(*
  This StartPosDetect supports different modes:
  - Triangle Markus
  - Internal StartPos generation (simulation based on substrate length and gap)
*)
FUNCTION_BLOCK FB_StartPositionWeu EXTENDS T_NamedBase IMPLEMENTS I_StartPosDetect
VAR_INPUT
  bEnable                         : BOOL;            // enable start position detection
  nCurrentPos                     : DINT;            // current position in Pulses/Subpixels
  fCurrentSpeed                   : LREAL;           // actual speed of conveyor in [m/s]
  fSubstrateLength                : LREAL;           // substrate length in [m]
  bUseExternalStartPos            : BOOL;            // Use external start position source
END_VAR
VAR_OUTPUT
  fLateralOffset                  : LREAL;           // Lateral +/- shift in Y [m]
  fSubstrateLengthDetected        : LREAL;           // Detected substrate length
  nPrintMarkPosBits               : WORD;            // Print mark position (bit coded),  TODO: avoid this specific code
END_VAR
VAR
  bInit : BOOL;   // fb initialized
  nMode : (MARK, SIMULATE_INTERN, SIMULATE_EXTERN) := MARK;   // StartTrigger mode
  
  // config
  _fResolutionPrint : LREAL;
  _fResolutionSubPx : LREAL;
  _pMarkDefinition : POINTER TO ST_MarkDefinition_Triangle;
  _iStartPosDetectExt : I_StartPosDetect;   // external start position source
   
  // instances
  fbMarkDetection : FB_MarkDetection_Triangle;    // StartPosition detection by marks
  fbStartPosSim   : FB_StartPositionDummy;        // StartPosition simulation

  // helper
  _bStart : BOOL;
  _nX0 : DINT;
  _bValid : BOOL;
  tOn_MissingMarksCheck : TON;   // trigger check (triggers within given time)
END_VAR

// TODO: >>>>>>>>>>>>>>>>>>>>>>>>>>>>>>>>>>>
// (optional) Mode: Encoder C HW_LATCH instead of marks
// <<<<<<<<<<<<<<<<<<<<<<<<<<<<<<<<<<<<<<<<<

// check parameter
IF NOT bInit THEN RETURN; END_IF
IF fCurrentSpeed = 0 THEN RETURN ; END_IF   // avoid 0 division

// default values (outputs and properties)
_bStart := FALSE;
_bValid := TRUE;
nPrintMarkPosBits := 0;  // no marks used
fLateralOFfset := 0;
fSubstrateLengthDetected := fSubstrateLength;

// mode selection
IF _pMarkDefinition = 0 OR_ELSE NOT _pMarkDefinition^.bEnabled THEN
  nMode :=  SEL(bUseExternalStartPos AND _iStartPosDetectExt <> 0, 
                  SIMULATE_INTERN, 
                  SIMULATE_EXTERN
                );
ELSIF NOT _pMarkDefinition^.bEnabled THEN   // if mark config is given and enabled
  nMode := MARK; 
END_IF

// run mode
IF nMode = MARK  THEN 
  // - with mark (forward / backward / other mark orientation)
  fbMarkDetection(
    bEnable:=bEnable,
    fResolution:=_fResolutionPrint*_fResolutionSubPx,
    fSubstrateLength:=fSubstrateLength,
    pMarkDefinition:=_pMarkDefinition,
    nCurrentPos:=nCurrentPos,
    fCurrentSpeed:=fCurrentSpeed,
    //bStartTrig=>_bStart,
    //nOffset_X0=>_nX0,
    fLateralOffset=>fLateralOffset,
    fSubstrateLengthDetected=>fSubstrateLengthDetected
  );
  // set I_StartPosDetect properties
  _bStart := fbMarkDetection.bStartTrig;
  _bValid := TRUE;
  _nX0    := fbMarkDetection.nOffset_X0;
  
 (*Check area with the correct arrangement of the mark sensor*)
 IF fbMarkDetection.bAreaOk THEN nPrintMarkPosBits.2 := TRUE; (*mark position in center*) 
  ELSIF fbMarkDetection.fLateralOffset > 0  THEN nPrintMarkPosBits.1 := TRUE; (*mark position on side I*) 
  ELSIF fbMarkDetection.fLateralOffset < 0  THEN nPrintMarkPosBits.3 := TRUE; (*mark position on side II*) 
  END_IF
  
  
ELSIF nMode = SIMULATE_INTERN THEN
  // without mark, simulate internally, started by external trigger and re-occur after every image/sheet length
  fbStartPosSim.bEnable := bEnable;                     // start simulatin with enable
  fbStartPosSim.bAutoTrigger := TRUE;
  fbStartPosSim.fSheetGap := 0;
  fbStartPosSim.fSubstrateLength := fSubstrateLength;   // same as given
  fbStartPosSim(
    //bTrigger:=,
    lPosition:=nCurrentPos,
    fSpeed:=fCurrentSpeed,
    fResolution:=_fResolutionPrint*_fResolutionSubPx
  );
  // set I_StartPosDetect properties
  _bStart := fbStartPosSim.bStartTrig;
  _bValid := fbStartPosSim.bValid;
  _nX0    := fbStartPosSim.nStartPositionX0;
  
  
ELSIF nMode = SIMULATE_EXTERN THEN
  // without mark, based on external reference
  
  // set I_StartPosDetect properties
  _bStart := ;
  _bValid := TRUE;
  _nX0    := ;
ELSE
  ;
END_IF


// supervision of mark missing (at least one trigger within 2 image lengths
//     nPrintMarkPosBits.0 := TRUE; (*=1 mark missing*) 
tOn_MissingMarksCheck(IN := bEnable AND NOT _bStart, PT := REAL_TO_TIME((2 * fSubstrateLength) / fCurrentSpeed * 1000), 
                      Q=>nPrintMarkPosBits.0
);

{warning 'add property implementation'}
(*
  A new container detected.
  NOTE: a pulse only
*)
PROPERTY bStartTrig : BOOL
GET
bStartTrig := _bStart;
END_GET
END_PROPERTY

{warning 'add property implementation'}
(*
  A valid container detected.
*)
PROPERTY bValid : BOOL
GET
bValid := _bValid;
END_GET
END_PROPERTY

METHOD Init
VAR_INPUT
  fPrintResolution      : LREAL := 600;         // print(head) resolution in [dpi]
  fSubPxResolution      : LREAL := 32;          // SubPixel resolution [SubPx], resolution factor (fI_PrintResolution*fI_SubPxResolution=>Output resolution)
  pMarkDefinition       : POINTER TO ST_MarkDefinition_Triangle;
  iStartPosDetectExt     : I_StartPosDetect;   // external start position source
END_VAR
IF _pMarkDefinition = 0 THEN LogError('Invalid parameter'); END_IF

_fResolutionPrint := fPrintResolution;
_fResolutionSubPx := fSubPxResolution;
_pMarkDefinition := pMarkDefinition;
_iStartPosDetectExt := iStartPosDetectExt;

// (optional) we use pointerTo_PU.registerStatusClient(sClient := fbStartPosSim);

bInit := TRUE;
END_METHOD

{warning 'add property implementation'}
(*
  Detected start position X0 (absolute) in [SubPx].
*)
PROPERTY nStartPositionX0 : DINT
GET
nStartPositionX0 := _nX0;
END_GET
END_PROPERTY

METHOD reset
fbMarkDetection.reset();
END_METHOD

END_FUNCTION_BLOCK

(* stored: Version 1.1.0.1, ProductVersion 3.1.4024.11
   POU FB_StartPositionWeu: Id {57e46adf-0651-4188-b0a4-ce8ff8a13827}, SpecialFunc None
   Folder I_StartPosDetect: Id {3bb3d753-1c9e-472a-8c3f-aec14f002339}
   Property bStartTrig: Id {e283e51a-7bd3-43b7-929a-8344709bc1e4}
   Get Get: Id {d88d396b-d2d9-47aa-81b3-e6702f1b2da2}
   Property bValid: Id {41d06b7b-92f2-4bfb-b40f-9ec4299b6723}
   Get Get: Id {b92c99f7-0a7d-43bc-bf16-56f41d6ca946}
   Method Init: Id {01bf650e-7028-4cf6-a973-171d14a98e24}
   Property nStartPositionX0: Id {06a37ff4-d366-43a1-82a9-5e3599c3a8b1}
   Get Get: Id {f436fe25-f2e2-42fc-baef-e97b91a2c4cc}
   Method Reset: Id {d27785f9-97b4-40ba-9b2e-a44c292ce0d7} *)
